INTERFACE itfSynchronizedAxisCommand EXTENDS itfAxisCommand

PROPERTY InSync : BOOL
GET
END_GET
END_PROPERTY

END_INTERFACE

(* stored: Version 1.1.0.1, ProductVersion 3.1.4024.12
   Itf itfSynchronizedAxisCommand: Id {62442c67-c113-4a02-9462-5fd7509e10b4}
   Property InSync: Id {02778b28-79c9-4fc0-9001-c310370018b4}
   Get Get: Id {b3470ea2-1c29-45cd-a5f7-06844eb77f19} *)
